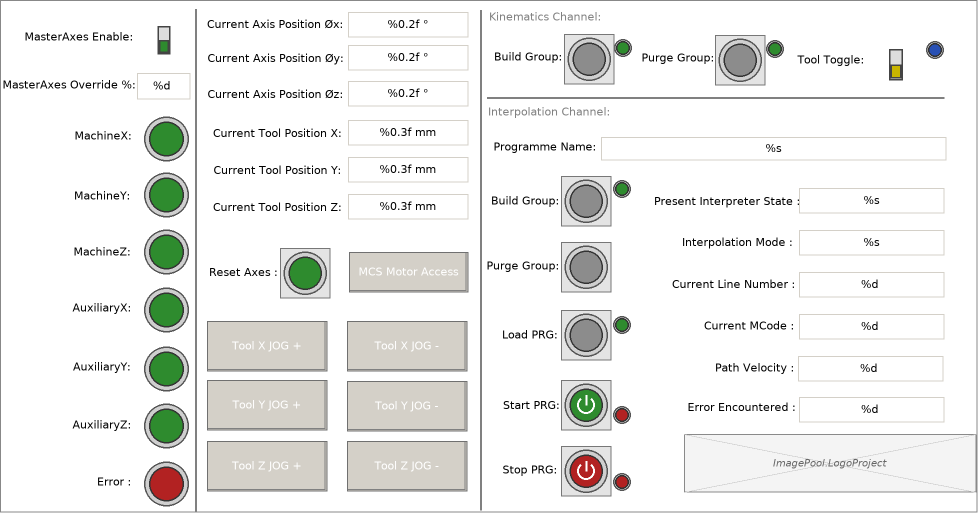
VISUALIZATION CtrlPANEL  // 978x513
    Lamp1 (137,113 59x52), variable: out_bMachX_Status, style: Lamp-Lamp1-Green
    Lamp1 (137,226 59x52), variable: out_bMachZ_Status, style: Lamp-Lamp1-Green
    Lamp1 (137,169 59x52), variable: out_bMachY_Status, style: Lamp-Lamp1-Green
    Lamp1 (137,284 59x52), variable: out_bSimsX_Status, style: Lamp-Lamp1-Green
    Lamp1 (137,343 59x52), variable: out_bSimsY_Status, style: Lamp-Lamp1-Green
    Lamp1 (137,400 59x52), variable: out_bSimsZ_Status, style: Lamp-Lamp1-Green
    DipSwitch (134,26 60x28), variable: in_bMasterAxes_Enable, behaviour: TOGGLE, style: Switch-DipSwitch-Green
    Line (196,511) (196,9)
    Label (65,121 76x30), "MachineX:"
    Label (64,181 76x30), "MachineY:"
    Label (64,237 76x30), "MachineZ:"
    Label (64,293 76x30), "AuxiliaryX:"
    Label (64,352 76x30), "AuxiliaryY:"
    Label (64,410 76x30), "AuxiliaryZ:"
    Label (19,22 120x30), "MasterAxes Enable:"
    Label (4,70 130x30), "MasterAxes Override %:"
    Button (207,321 120x50), "Tool X JOG +"
        tap in_bAxes_SimsX_Jog_Forward
    Button (207,380 120x50), "Tool Y JOG +"
        tap in_bAxes_SimsY_Jog_Forward
    Button (207,441 120x50), "Tool Z JOG +"
        tap in_bAxes_SimsZ_Jog_Forward
    Button (347,321 120x50), "Tool X JOG -"
        tap in_bAxes_SimsX_Jog_Backward
    Button (347,381 120x50), "Tool Y JOG -"
        tap in_bAxes_SimsY_Jog_Backward
    Textfield (348,12 120x25), "%0.2f °", text variable: MachX.NcToPlc.ActPos
    Textfield (348,45 120x25), "%0.2f °", text variable: MachY.NcToPlc.ActPos
    Textfield (348,81 120x25), "%0.2f °", text variable: MachZ.NcToPlc.ActPos
    Textfield (348,120 120x25), "%0.3f mm", text variable: SimsX.NcToPlc.ActPos
    Textfield (348,157 120x25), "%0.3f mm", text variable: SimsY.NcToPlc.ActPos
    Textfield (348,194 120x25), "%0.3f mm", text variable: SimsZ.NcToPlc.ActPos
    Label (211,119 133x29), "Current Tool Position X:"
    Label (211,156 133x29), "Current Tool Position Y:"
    Label (211,193 133x29), "Current Tool Position Z:"
    Label (205,10 140x29), "Current Axis Position Øx:"
    Label (209,44 133x29), "Current Axis Position Øy:"
    Label (209,80 133x29), "Current Axis Position Øz:"
    Line (481,510) (481,10)
    Button (347,441 120x50), "Tool Z JOG -"
        tap in_bAxes_SimsZ_Jog_Backward
    Label (460,42 136x30), "Build Group:"
    Lamp1 (613,38 20x20), variable: out_bAxes_KinConfigGroup_Done_HMI, style: Lamp-Lamp1-Green
    Label (619,41 118x34), "Purge Group:"
    PushSwitch (715,35 50x50), variable: in_bAxes_KinResetGroup_Execute, behaviour: TAP, style: Switch-PushSwitch-Gray
    Lamp1 (765,39 20x20), variable: out_bAxes_KinResetGroup_Done, style: Lamp-Lamp1-Green
    Line (944,98) (487,98)
    Label (477,2 136x30), "Kinematics Channel:"
    Label (481,97 136x30), "Interpolation Channel:"
    PushSwitch (561,310 50x50), variable: in_bAxes_ItpLoadPRG_Execute, behaviour: TOGGLE, style: Switch-PushSwitch-Gray
    Lamp1 (612,405 20x20), variable: in_bAxes_ItpStartStop_Error, style: Lamp-Lamp1-Red
    Label (457,186 136x30), "Build Group:"
    Label (462,320 136x30), "Load PRG:"
    Label (464,390 135x31), "Start PRG:"
    Label (462,455 136x30), "Stop PRG:"
    Lamp1 (612,472 20x20), variable: in_bAxes_ItpStartStop_Error, style: Lamp-Lamp1-Red
    Label (477,132 136x30), "Programme Name:"
    Textfield (601,137 345x23), "%s", tooltip "Please Enter the .nc file Path Here", text variable: in_strAxes_ItpLoadPRG_PRGPath
        OnMouseClick: write in_strAxes_ItpLoadPRG_PRGPath via VisuDialogs.Keypad
    Textfield (137,73 53x26), "%d", text variable: in_uiMasterAxes_Override
        OnMouseClick: write the text variable via VisuDialogs.Numpad
    Lamp1 (612,179 20x20), variable: out_bAxes_BuildItpGoup_Done, style: Lamp-Lamp1-Green
    DipSwitch (866,49 60x31), variable: in_bTOOL, behaviour: TOGGLE, style: Switch-DipSwitch-Yellow
    Lamp1 (925,40 20x20), variable: out_bTOOL_HW, style: Lamp-Lamp1-Blue
    Label (763,45 136x30), "Tool Toggle:"
    Lamp1 (137,458 59x52), variable: out_bAxes_Master_Error, style: Lamp-Lamp1-Red
    Label (76,467 76x30), "Error :"
    Textfield (799,188 145x25), "%s", text variable: out_stItp_InterpreterState_String
    Label (657,187 140x29), "Present Interpreter State :"
    Textfield (799,230 145x25), "%s", text variable: out_wdItp_InterpolationMode_string
    Label (667,228 141x29), "Interpolation Mode :"
    Textfield (799,272 145x25), "%d", text variable: out_uiItp_Linenumber
    Label (669,270 129x29), "Current Line Number :"
    Textfield (799,314 145x25), "%d", text variable: out_uiItp_Mcodenumber
    Label (702,312 94x28), "Current MCode :"
    Textfield (799,397 145x25), "%d", text variable: out_uiItp_ErrorEncountered
    Label (690,393 103x29), "Error Encountered :"
    Textfield (798,356 145x25), "%d", text variable: out_uiItp_Feedrate
    Label (708,354 93x28), "Path Velocity :"
    PushSwitch (561,242 50x50), variable: in_bAxes_ItpReConfig_Group_Execute, behaviour: TAP, style: Switch-PushSwitch-Gray
    Label (455,251 136x30), "Purge Group:"
    PushSwitch (564,34 50x50), variable: in_bAxes_KinConfigGroup_Execute, behaviour: TAP, style: Switch-PushSwitch-Gray
    PushSwitch (561,176 50x50), variable: in_bAxes_BuildItpGoup_Execute, behaviour: TOGGLE, style: Switch-PushSwitch-Gray
    PowerSwitch (561,380 50x50), variable: in_bAxes_ItpStartStop_Start, behaviour: TOGGLE, style: Switch-PowerSwitch-Green
    PowerSwitch (561,446 50x50), variable: in_bAxes_ItpStartStop_Stop, behaviour: TOGGLE, style: Switch-PowerSwitch-Red
    Lamp1 (612,315 20x20), variable: out_bAxes_ItpLoadPRG_DoneHMI, style: Lamp-Lamp1-Green
    Button (349,252 119x40), "MCS Motor Access"
        toggle in_b_MoveHome
        OnMouseClick: OpenDialog Dialog=Home, OpenModal=True, OpenCentered=True
    PushSwitch (280,248 50x50), variable: Axes_Reset_All, behaviour: TAP, style: Switch-PushSwitch-Green
    Label (192,258 103x29), "Reset Axes :"
    Image (684,434 292x58), image: ImagePool.LogoProject
END_VISUALIZATION

(* stored: Version 1.1.0.1, ProductVersion 3.1.4022.17
   Visu CtrlPANEL: Id {f1fba6ff-2e8e-4df3-ae8b-4b25dd87c5f2} *)
